(* CODESYS project T1_Simple.project

Project tree, tasks and I/O mapping:
  Device : CODESYS Control Win V3, 3S - Smart Software Solutions GmbH, order no. 305021, version 3.5.7.20
    application Application
      libraries: Standard, * (System); Util, * (System)
      task MainTask (cyclic, interval t#20ms, priority 1) calls PLC_PRG
      program PLC_PRG [FBD]
      global variables GVL
      Symbols
*)

// Device/Application/GVL
VAR_GLOBAL
	PV_h: REAL;
	SP_h: REAL;
	h_man: REAL;
	u1_man: REAL;
	MAN: BOOL;
	RES: BOOL;
	u1_h: REAL;
	SP_t: REAL;
	PV_t: REAL;
	u2_man: REAL;
	RES_u2: BOOL;
	u2_h: REAL;
	Kp_h: REAL;
	TN_h: REAL;
	TV_h: REAL;
	KP_t: REAL;
	TN_t: REAL;
	TV_t: REAL;
END_VAR

// Device/Application/PLC_PRG
PROGRAM PLC_PRG
VAR
	PID_H: PID;
	PID_T: PID;
END_VAR

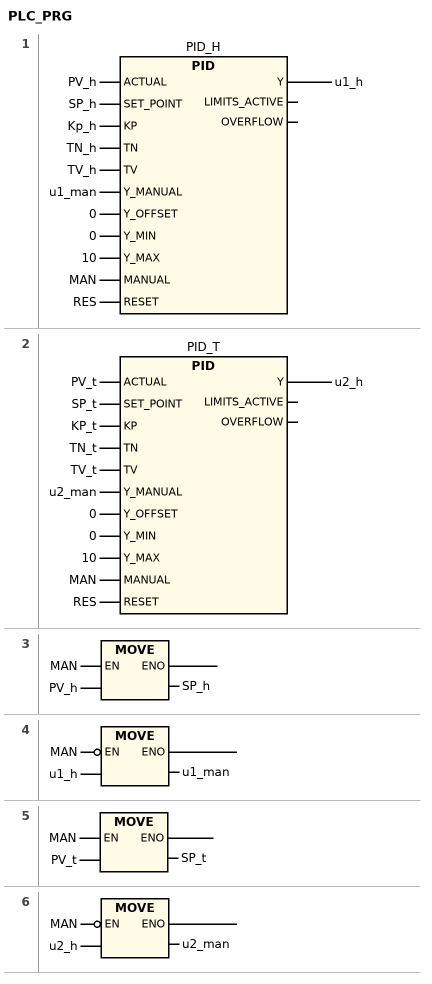
// NETWORK 1
PID_H(
    ACTUAL := PV_h,
    SET_POINT := SP_h,
    KP := Kp_h,
    TN := TN_h,
    TV := TV_h,
    Y_MANUAL := u1_man,
    Y_OFFSET := 0,
    Y_MIN := 0,
    Y_MAX := 10,
    MANUAL := MAN,
    RESET := RES); // PID
u1_h := PID_H.Y;

// NETWORK 2
PID_T(
    ACTUAL := PV_t,
    SET_POINT := SP_t,
    KP := KP_t,
    TN := TN_t,
    TV := TV_t,
    Y_MANUAL := u2_man,
    Y_OFFSET := 0,
    Y_MIN := 0,
    Y_MAX := 10,
    MANUAL := MAN,
    RESET := RES); // PID
u2_h := PID_T.Y;

// NETWORK 3
IF MAN THEN SP_h := PV_h; END_IF

// NETWORK 4
IF NOT MAN THEN u1_man := u1_h; END_IF

// NETWORK 5
IF MAN THEN SP_t := PV_t; END_IF

// NETWORK 6
IF NOT MAN THEN u2_man := u2_h; END_IF

END_PROGRAM
